{region '#Template'}
	{attribute 'Version' := '5.0.0.0'}
	{attribute 'Tags' := '"LCID": "1031", "Text": "AC, Allgemein, AHU, Priorität"'}
	{attribute 'Tags' := '"LCID": "1033", "Text": "AC, General, AHU, Priority"'}
	{attribute 'Using' := '"Type": "Template", "URI": "E_BA_AC_OpMod01"'}
	{attribute 'Description' := '"LCID": "1031", "Text": "Freigabe Prioritäten"'}
	{attribute 'Description' := '"LCID": "1033", "Text": "Enable priorities"'}
{endregion}
FUNCTION_BLOCK FB_BA_AC_EnPrio
VAR_INPUT
	eOpMode					: E_BA_AC_OpMod01;
END_VAR
VAR_OUTPUT
	stPriorityEn			: ST_BA_PriorityEn;
END_VAR
VAR
	PrioSwiPlt				: FB_BA_MMUX_B24;
	PrioSwiSfty				: FB_BA_MMUX_B08;
	PrioSwiCrit				: FB_BA_MMUX_B08;
	PrioSwiPgm				: FB_BA_MMUX_B08;
END_VAR

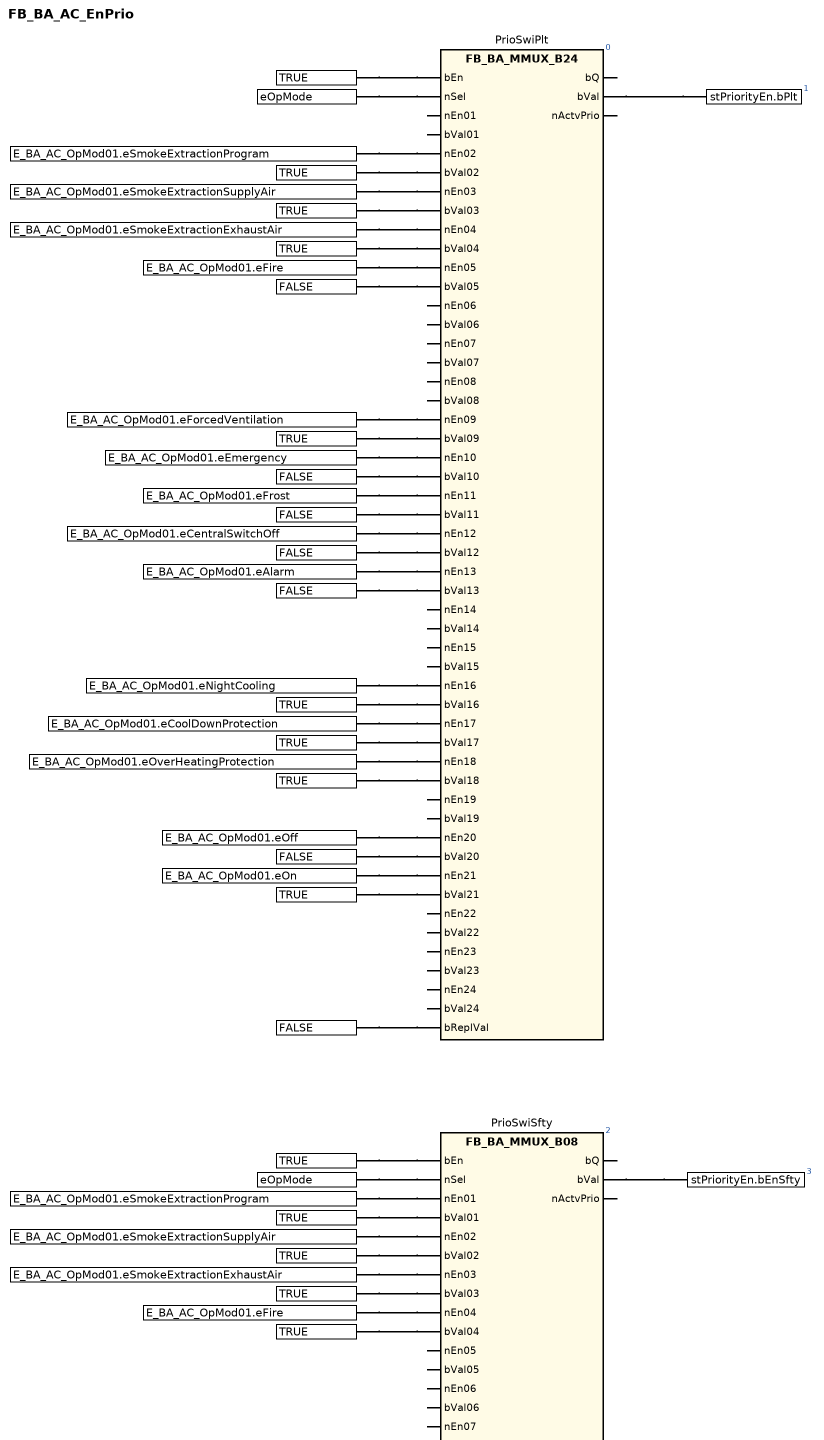
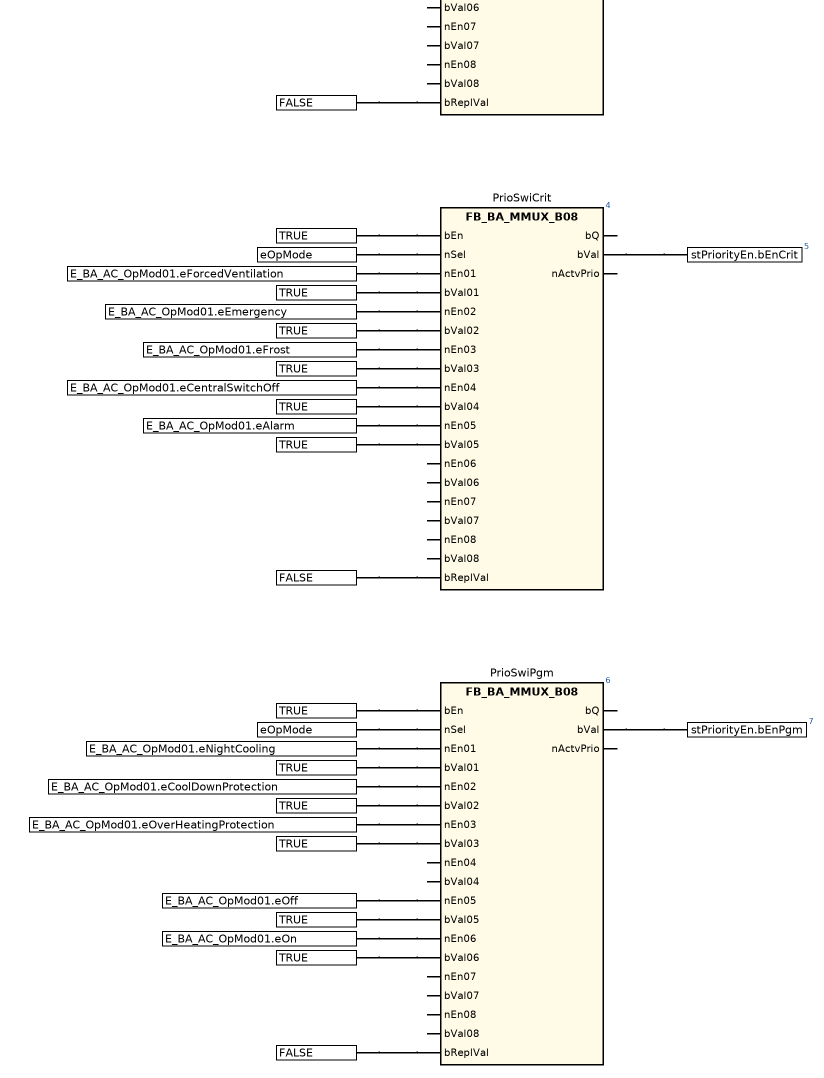
PrioSwiPlt(
    bEn := TRUE,
    nSel := eOpMode,
    nEn02 := E_BA_AC_OpMod01.eSmokeExtractionProgram,
    bVal02 := TRUE,
    nEn03 := E_BA_AC_OpMod01.eSmokeExtractionSupplyAir,
    bVal03 := TRUE,
    nEn04 := E_BA_AC_OpMod01.eSmokeExtractionExhaustAir,
    bVal04 := TRUE,
    nEn05 := E_BA_AC_OpMod01.eFire,
    bVal05 := FALSE,
    nEn09 := E_BA_AC_OpMod01.eForcedVentilation,
    bVal09 := TRUE,
    nEn10 := E_BA_AC_OpMod01.eEmergency,
    bVal10 := FALSE,
    nEn11 := E_BA_AC_OpMod01.eFrost,
    bVal11 := FALSE,
    nEn12 := E_BA_AC_OpMod01.eCentralSwitchOff,
    bVal12 := FALSE,
    nEn13 := E_BA_AC_OpMod01.eAlarm,
    bVal13 := FALSE,
    nEn16 := E_BA_AC_OpMod01.eNightCooling,
    bVal16 := TRUE,
    nEn17 := E_BA_AC_OpMod01.eCoolDownProtection,
    bVal17 := TRUE,
    nEn18 := E_BA_AC_OpMod01.eOverHeatingProtection,
    bVal18 := TRUE,
    nEn20 := E_BA_AC_OpMod01.eOff,
    bVal20 := FALSE,
    nEn21 := E_BA_AC_OpMod01.eOn,
    bVal21 := TRUE,
    bReplVal := FALSE); // FB_BA_MMUX_B24
stPriorityEn.bPlt := PrioSwiPlt.bVal;
PrioSwiSfty(
    bEn := TRUE,
    nSel := eOpMode,
    nEn01 := E_BA_AC_OpMod01.eSmokeExtractionProgram,
    bVal01 := TRUE,
    nEn02 := E_BA_AC_OpMod01.eSmokeExtractionSupplyAir,
    bVal02 := TRUE,
    nEn03 := E_BA_AC_OpMod01.eSmokeExtractionExhaustAir,
    bVal03 := TRUE,
    nEn04 := E_BA_AC_OpMod01.eFire,
    bVal04 := TRUE,
    bReplVal := FALSE); // FB_BA_MMUX_B08
stPriorityEn.bEnSfty := PrioSwiSfty.bVal;
PrioSwiCrit(
    bEn := TRUE,
    nSel := eOpMode,
    nEn01 := E_BA_AC_OpMod01.eForcedVentilation,
    bVal01 := TRUE,
    nEn02 := E_BA_AC_OpMod01.eEmergency,
    bVal02 := TRUE,
    nEn03 := E_BA_AC_OpMod01.eFrost,
    bVal03 := TRUE,
    nEn04 := E_BA_AC_OpMod01.eCentralSwitchOff,
    bVal04 := TRUE,
    nEn05 := E_BA_AC_OpMod01.eAlarm,
    bVal05 := TRUE,
    bReplVal := FALSE); // FB_BA_MMUX_B08
stPriorityEn.bEnCrit := PrioSwiCrit.bVal;
PrioSwiPgm(
    bEn := TRUE,
    nSel := eOpMode,
    nEn01 := E_BA_AC_OpMod01.eNightCooling,
    bVal01 := TRUE,
    nEn02 := E_BA_AC_OpMod01.eCoolDownProtection,
    bVal02 := TRUE,
    nEn03 := E_BA_AC_OpMod01.eOverHeatingProtection,
    bVal03 := TRUE,
    nEn05 := E_BA_AC_OpMod01.eOff,
    bVal05 := TRUE,
    nEn06 := E_BA_AC_OpMod01.eOn,
    bVal06 := TRUE,
    bReplVal := FALSE); // FB_BA_MMUX_B08
stPriorityEn.bEnPgm := PrioSwiPgm.bVal;

END_FUNCTION_BLOCK

(* stored: Version 1.1.0.1, ProductVersion 3.1.4024.12
   POU FB_BA_AC_EnPrio: Id {f913e6b4-eed0-4451-9836-e9b69a4d2575}, SpecialFunc None *)
